// TIA Portal V19 export
FUNCTION_BLOCK "ValveMachine_FB"   // FB125, LAD
TITLE = VALVE MACHINE
// stored: Access Published, MemoryReserve 100, SetENOAutomatically false
   VAR_INPUT
      AreaInterface : "AreaInterface";
      ZSI : "udt_ZoneSafetyInterface";
      DSI : "udt_DeviceSafetyInterface";
      DataIn : "ValveMachine_DataIn";
      Cin : "ValveMachine_Cin";
      Config : "ValveMachine_Config";
   END_VAR
   VAR_OUTPUT
      MachineInterface : "MachineInterface";
      COut : "ValveMachine_COut";
      DataOut : "ValveMachine_DataOut";
   END_VAR
   VAR_IN_OUT
      Alarm : "ValveAlr";
      Warning : "ValveMachine_Wng";
   END_VAR
   VAR
      Sts : Struct
         Standstill : Bool;
         AlarmsPresence : Bool;
         WarningsPresence : Bool;
         Rest_Cnd : Bool;
         Work_Cnd : Bool;
      END_STRUCT;
      Ctrl : Struct
         StopDueDoorOpeningRequest : Bool;
         StopInPhase : Bool;
         StopProgrammed : Bool;
         StopAborting : Bool;
         Work : Bool;
         Rest : Bool;
         Rest_Man : Bool;
         Work_Man : Bool;
         Rest_Aut : Bool;
         Work_Aut : Bool;
      END_STRUCT;
      V : "Valve";
      TON_NoPendingCmd : TON_TIME;
      TON_Rest_MissingExtEnable : TON_TIME;
      TON_Work_MissingExtEnable : TON_TIME;
      TON_PressureRunning_Timeout { S7_SetPoint := 'True'} : TON_TIME;
      Aux : Struct
         Pb_Rest : Bool;
         Pb_Work : Bool;
         Pb_StartStop : Bool;
      END_STRUCT;
   END_VAR
   VAR_TEMP
      PE : Struct
         Pb_Rest : Bool;
         Pb_Work : Bool;
         Pb_StartStop : Bool;
      END_STRUCT;
   END_VAR
   VAR_TEMP   // added for the SCL form of the ladder/FBD networks
      _w1 : Bool;
      _w2 : Bool;
      _w3 : Bool;
   END_VAR
BEGIN

REGION Network 1: Positive edges
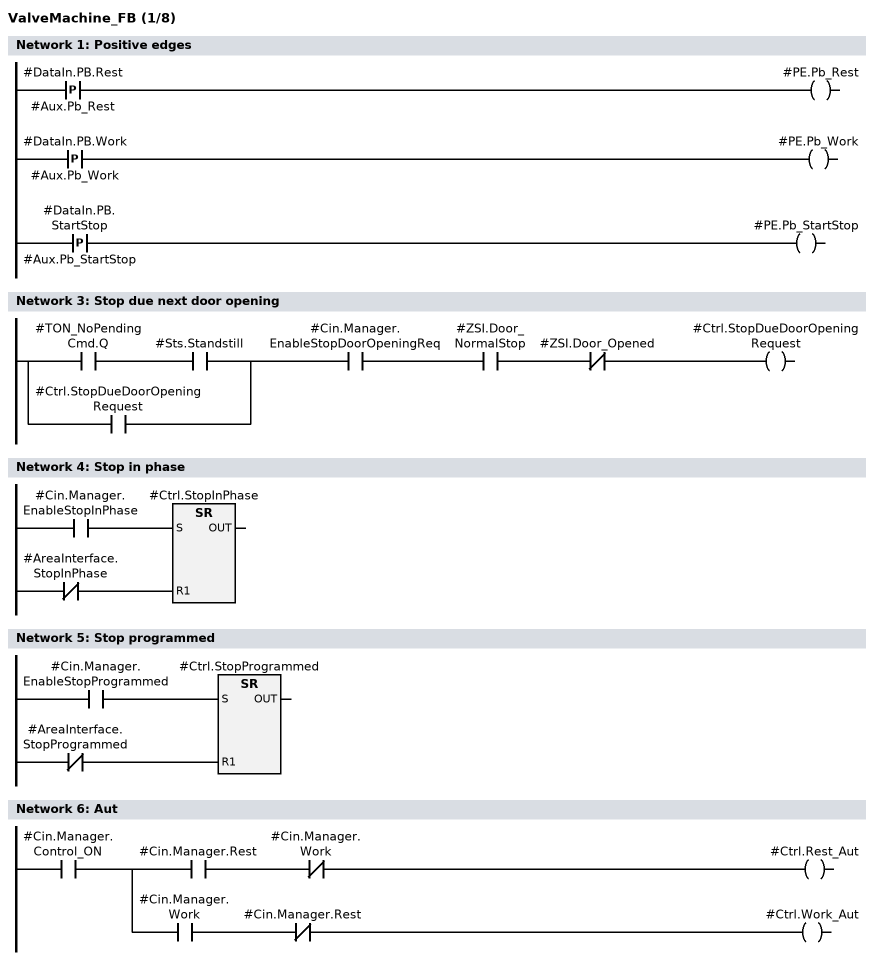
   RUNG wire#powerrail
      P_Contact(operand := #DataIn.PB.Rest, bit := #Aux.Pb_Rest)
      Coil( #PE.Pb_Rest )
   END_RUNG
   RUNG wire#powerrail
      P_Contact(operand := #DataIn.PB.Work, bit := #Aux.Pb_Work)
      Coil( #PE.Pb_Work )
   END_RUNG
   RUNG wire#powerrail
      P_Contact(operand := #DataIn.PB.StartStop, bit := #Aux.Pb_StartStop)
      Coil( #PE.Pb_StartStop )
   END_RUNG
   // the same network as SCL:
   #_w1 := #DataIn.PB.Rest AND NOT #Aux.Pb_Rest;   // rising edge of #DataIn.PB.Rest
   #Aux.Pb_Rest := #DataIn.PB.Rest;
   #PE.Pb_Rest := #_w1;
   #_w2 := #DataIn.PB.Work AND NOT #Aux.Pb_Work;   // rising edge of #DataIn.PB.Work
   #Aux.Pb_Work := #DataIn.PB.Work;
   #PE.Pb_Work := #_w2;
   #_w3 := #DataIn.PB.StartStop AND NOT #Aux.Pb_StartStop;   // rising edge of #DataIn.PB.StartStop
   #Aux.Pb_StartStop := #DataIn.PB.StartStop;
   #PE.Pb_StartStop := #_w3;
END_REGION

REGION Network 2: <<< MACHINE STOP >>>
END_REGION

REGION Network 3: Stop due next door opening
   RUNG wire#powerrail
      Contact( #TON_NoPendingCmd.Q )
      Contact( #Sts.Standstill )
      wire#w1
      Contact( #Cin.Manager.EnableStopDoorOpeningReq )
      Contact( #ZSI.Door_NormalStop )
      I_Contact( #ZSI.Door_Opened )
      Coil( #Ctrl.StopDueDoorOpeningRequest )
   END_RUNG
   RUNG wire#powerrail
      Contact( #Ctrl.StopDueDoorOpeningRequest )
   END_RUNG wire#w1
   // the same network as SCL:
   #Ctrl.StopDueDoorOpeningRequest := ((#TON_NoPendingCmd.Q AND #Sts.Standstill) OR #Ctrl.StopDueDoorOpeningRequest) AND #Cin.Manager.EnableStopDoorOpeningReq AND #ZSI.Door_NormalStop AND NOT #ZSI.Door_Opened;
END_REGION

REGION Network 4: Stop in phase
   RUNG wire#powerrail
      Contact( #Cin.Manager.EnableStopInPhase )
      S_SR(operand := #Ctrl.StopInPhase, r1 := wire#w1)
   END_RUNG
   RUNG wire#powerrail
      I_Contact( #AreaInterface.StopInPhase )
   END_RUNG wire#w1
   // the same network as SCL:
   IF #Cin.Manager.EnableStopInPhase THEN
       #Ctrl.StopInPhase := TRUE;   // SR flip-flop
   END_IF;
   IF NOT #AreaInterface.StopInPhase THEN #Ctrl.StopInPhase := FALSE; END_IF;
END_REGION

REGION Network 5: Stop programmed
   RUNG wire#powerrail
      Contact( #Cin.Manager.EnableStopProgrammed )
      S_SR(operand := #Ctrl.StopProgrammed, r1 := wire#w1)
   END_RUNG
   RUNG wire#powerrail
      I_Contact( #AreaInterface.StopProgrammed )
   END_RUNG wire#w1
   // the same network as SCL:
   IF #Cin.Manager.EnableStopProgrammed THEN
       #Ctrl.StopProgrammed := TRUE;   // SR flip-flop
   END_IF;
   IF NOT #AreaInterface.StopProgrammed THEN #Ctrl.StopProgrammed := FALSE; END_IF;
END_REGION

REGION Network 6: Aut
   RUNG wire#powerrail
      Contact( #Cin.Manager.Control_ON )
      wire#w1
      Contact( #Cin.Manager.Rest )
      I_Contact( #Cin.Manager.Work )
      Coil( #Ctrl.Rest_Aut )
   END_RUNG
   RUNG wire#w1
      Contact( #Cin.Manager.Work )
      I_Contact( #Cin.Manager.Rest )
      Coil( #Ctrl.Work_Aut )
   END_RUNG
   // the same network as SCL:
   #Ctrl.Rest_Aut := #Cin.Manager.Control_ON AND #Cin.Manager.Rest AND NOT #Cin.Manager.Work;
   #Ctrl.Work_Aut := #Cin.Manager.Control_ON AND #Cin.Manager.Work AND NOT #Cin.Manager.Rest;
END_REGION

REGION Network 7: Man
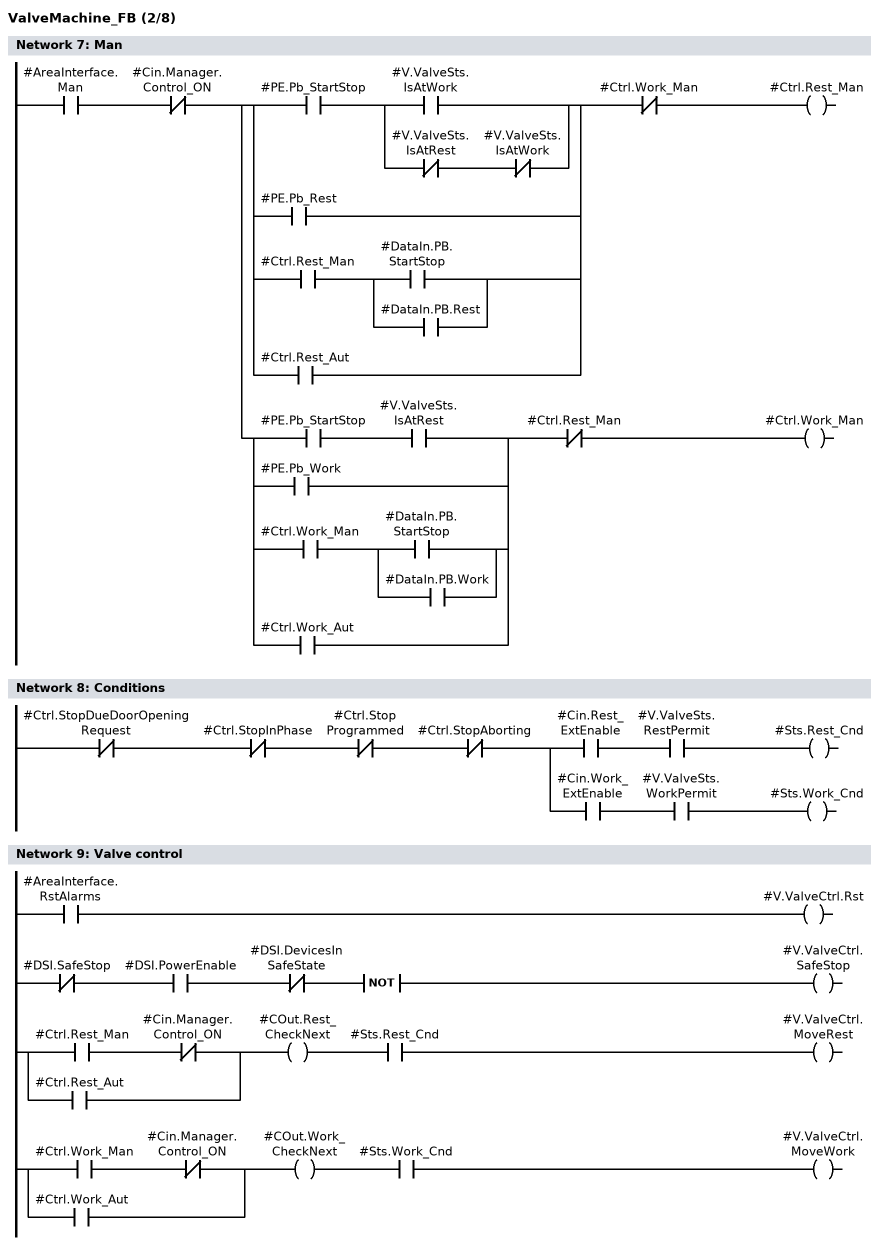
   RUNG wire#powerrail
      Contact( #AreaInterface.Man )
      I_Contact( #Cin.Manager.Control_ON )
      wire#w1
      Contact( #PE.Pb_StartStop )
      wire#w2
      Contact( #V.ValveSts.IsAtWork )
      wire#w3
      I_Contact( #Ctrl.Work_Man )
      Coil( #Ctrl.Rest_Man )
   END_RUNG
   RUNG wire#w2
      I_Contact( #V.ValveSts.IsAtRest )
      I_Contact( #V.ValveSts.IsAtWork )
   END_RUNG wire#w3
   RUNG wire#w1
      Contact( #PE.Pb_Rest )
   END_RUNG wire#w3
   RUNG wire#w1
      Contact( #Ctrl.Rest_Man )
      wire#w4
      Contact( #DataIn.PB.StartStop )
   END_RUNG wire#w3
   RUNG wire#w4
      Contact( #DataIn.PB.Rest )
   END_RUNG wire#w3
   RUNG wire#w1
      Contact( #Ctrl.Rest_Aut )
   END_RUNG wire#w3
   RUNG wire#w1
      Contact( #PE.Pb_StartStop )
      Contact( #V.ValveSts.IsAtRest )
      wire#w5
      I_Contact( #Ctrl.Rest_Man )
      Coil( #Ctrl.Work_Man )
   END_RUNG
   RUNG wire#w1
      Contact( #PE.Pb_Work )
   END_RUNG wire#w5
   RUNG wire#w1
      Contact( #Ctrl.Work_Man )
      wire#w6
      Contact( #DataIn.PB.StartStop )
   END_RUNG wire#w5
   RUNG wire#w6
      Contact( #DataIn.PB.Work )
   END_RUNG wire#w5
   RUNG wire#w1
      Contact( #Ctrl.Work_Aut )
   END_RUNG wire#w5
   // the same network as SCL:
   #_w1 := #AreaInterface.Man AND NOT #Cin.Manager.Control_ON;
   #Ctrl.Rest_Man := #_w1 AND ((#PE.Pb_StartStop AND (#V.ValveSts.IsAtWork OR (NOT #V.ValveSts.IsAtRest AND NOT #V.ValveSts.IsAtWork))) OR #PE.Pb_Rest OR (#Ctrl.Rest_Man AND (#DataIn.PB.StartStop OR #DataIn.PB.Rest)) OR #Ctrl.Rest_Aut) AND NOT #Ctrl.Work_Man;
   #Ctrl.Work_Man := #_w1 AND ((#PE.Pb_StartStop AND #V.ValveSts.IsAtRest) OR #PE.Pb_Work OR (#Ctrl.Work_Man AND (#DataIn.PB.StartStop OR #DataIn.PB.Work)) OR #Ctrl.Work_Aut) AND NOT #Ctrl.Rest_Man;
END_REGION

REGION Network 8: Conditions
   RUNG wire#powerrail
      I_Contact( #Ctrl.StopDueDoorOpeningRequest )
      I_Contact( #Ctrl.StopInPhase )
      I_Contact( #Ctrl.StopProgrammed )
      I_Contact( #Ctrl.StopAborting )
      wire#w1
      Contact( #Cin.Rest_ExtEnable )
      Contact( #V.ValveSts.RestPermit )
      Coil( #Sts.Rest_Cnd )
   END_RUNG
   RUNG wire#w1
      Contact( #Cin.Work_ExtEnable )
      Contact( #V.ValveSts.WorkPermit )
      Coil( #Sts.Work_Cnd )
   END_RUNG
   // the same network as SCL:
   #_w1 := NOT #Ctrl.StopDueDoorOpeningRequest AND NOT #Ctrl.StopInPhase AND NOT #Ctrl.StopProgrammed AND NOT #Ctrl.StopAborting;
   #Sts.Rest_Cnd := #_w1 AND #Cin.Rest_ExtEnable AND #V.ValveSts.RestPermit;
   #Sts.Work_Cnd := #_w1 AND #Cin.Work_ExtEnable AND #V.ValveSts.WorkPermit;
END_REGION

REGION Network 9: Valve control
   RUNG wire#powerrail
      Contact( #AreaInterface.RstAlarms )
      Coil( #V.ValveCtrl.Rst )
   END_RUNG
   RUNG wire#powerrail
      I_Contact( #DSI.SafeStop )
      Contact( #DSI.PowerEnable )
      I_Contact( #DSI.DevicesInSafeState )
      Not()
      Coil( #V.ValveCtrl.SafeStop )
   END_RUNG
   RUNG wire#powerrail
      Contact( #Ctrl.Rest_Man )
      I_Contact( #Cin.Manager.Control_ON )
      wire#w1
      Coil( #COut.Rest_CheckNext )
      Contact( #Sts.Rest_Cnd )
      Coil( #V.ValveCtrl.MoveRest )
   END_RUNG
   RUNG wire#powerrail
      Contact( #Ctrl.Rest_Aut )
   END_RUNG wire#w1
   RUNG wire#powerrail
      Contact( #Ctrl.Work_Man )
      I_Contact( #Cin.Manager.Control_ON )
      wire#w2
      Coil( #COut.Work_CheckNext )
      Contact( #Sts.Work_Cnd )
      Coil( #V.ValveCtrl.MoveWork )
   END_RUNG
   RUNG wire#powerrail
      Contact( #Ctrl.Work_Aut )
   END_RUNG wire#w2
   // the same network as SCL:
   #V.ValveCtrl.Rst := #AreaInterface.RstAlarms;
   #V.ValveCtrl.SafeStop := NOT (NOT #DSI.SafeStop AND #DSI.PowerEnable AND NOT #DSI.DevicesInSafeState);
   #COut.Rest_CheckNext := (#Ctrl.Rest_Man AND NOT #Cin.Manager.Control_ON) OR #Ctrl.Rest_Aut;
   #V.ValveCtrl.MoveRest := #COut.Rest_CheckNext AND #Sts.Rest_Cnd;
   #COut.Work_CheckNext := (#Ctrl.Work_Man AND NOT #Cin.Manager.Control_ON) OR #Ctrl.Work_Aut;
   #V.ValveCtrl.MoveWork := #COut.Work_CheckNext AND #Sts.Work_Cnd;
END_REGION

REGION Network 10: Warning missing external enables
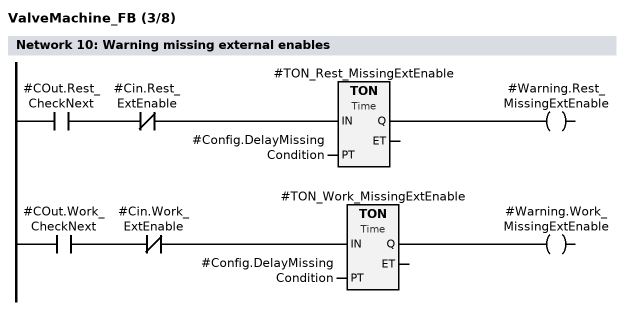
   RUNG wire#powerrail
      Contact( #COut.Rest_CheckNext )
      I_Contact( #Cin.Rest_ExtEnable )
      { S7_Templates := "time_type := Time" } #TON_Rest_MissingExtEnable.TON(pt := #Config.DelayMissingCondition, et =>)
      Coil( #Warning.Rest_MissingExtEnable )
   END_RUNG
   RUNG wire#powerrail
      Contact( #COut.Work_CheckNext )
      I_Contact( #Cin.Work_ExtEnable )
      { S7_Templates := "time_type := Time" } #TON_Work_MissingExtEnable.TON(pt := #Config.DelayMissingCondition, et =>)
      Coil( #Warning.Work_MissingExtEnable )
   END_RUNG
   // the same network as SCL:
   #TON_Rest_MissingExtEnable(IN := #COut.Rest_CheckNext AND NOT #Cin.Rest_ExtEnable,   // TON
                           PT := #Config.DelayMissingCondition);
   #Warning.Rest_MissingExtEnable := #TON_Rest_MissingExtEnable.Q;
   #TON_Work_MissingExtEnable(IN := #COut.Work_CheckNext AND NOT #Cin.Work_ExtEnable,   // TON
                           PT := #Config.DelayMissingCondition);
   #Warning.Work_MissingExtEnable := #TON_Work_MissingExtEnable.Q;
END_REGION

REGION Network 11: Valve manager
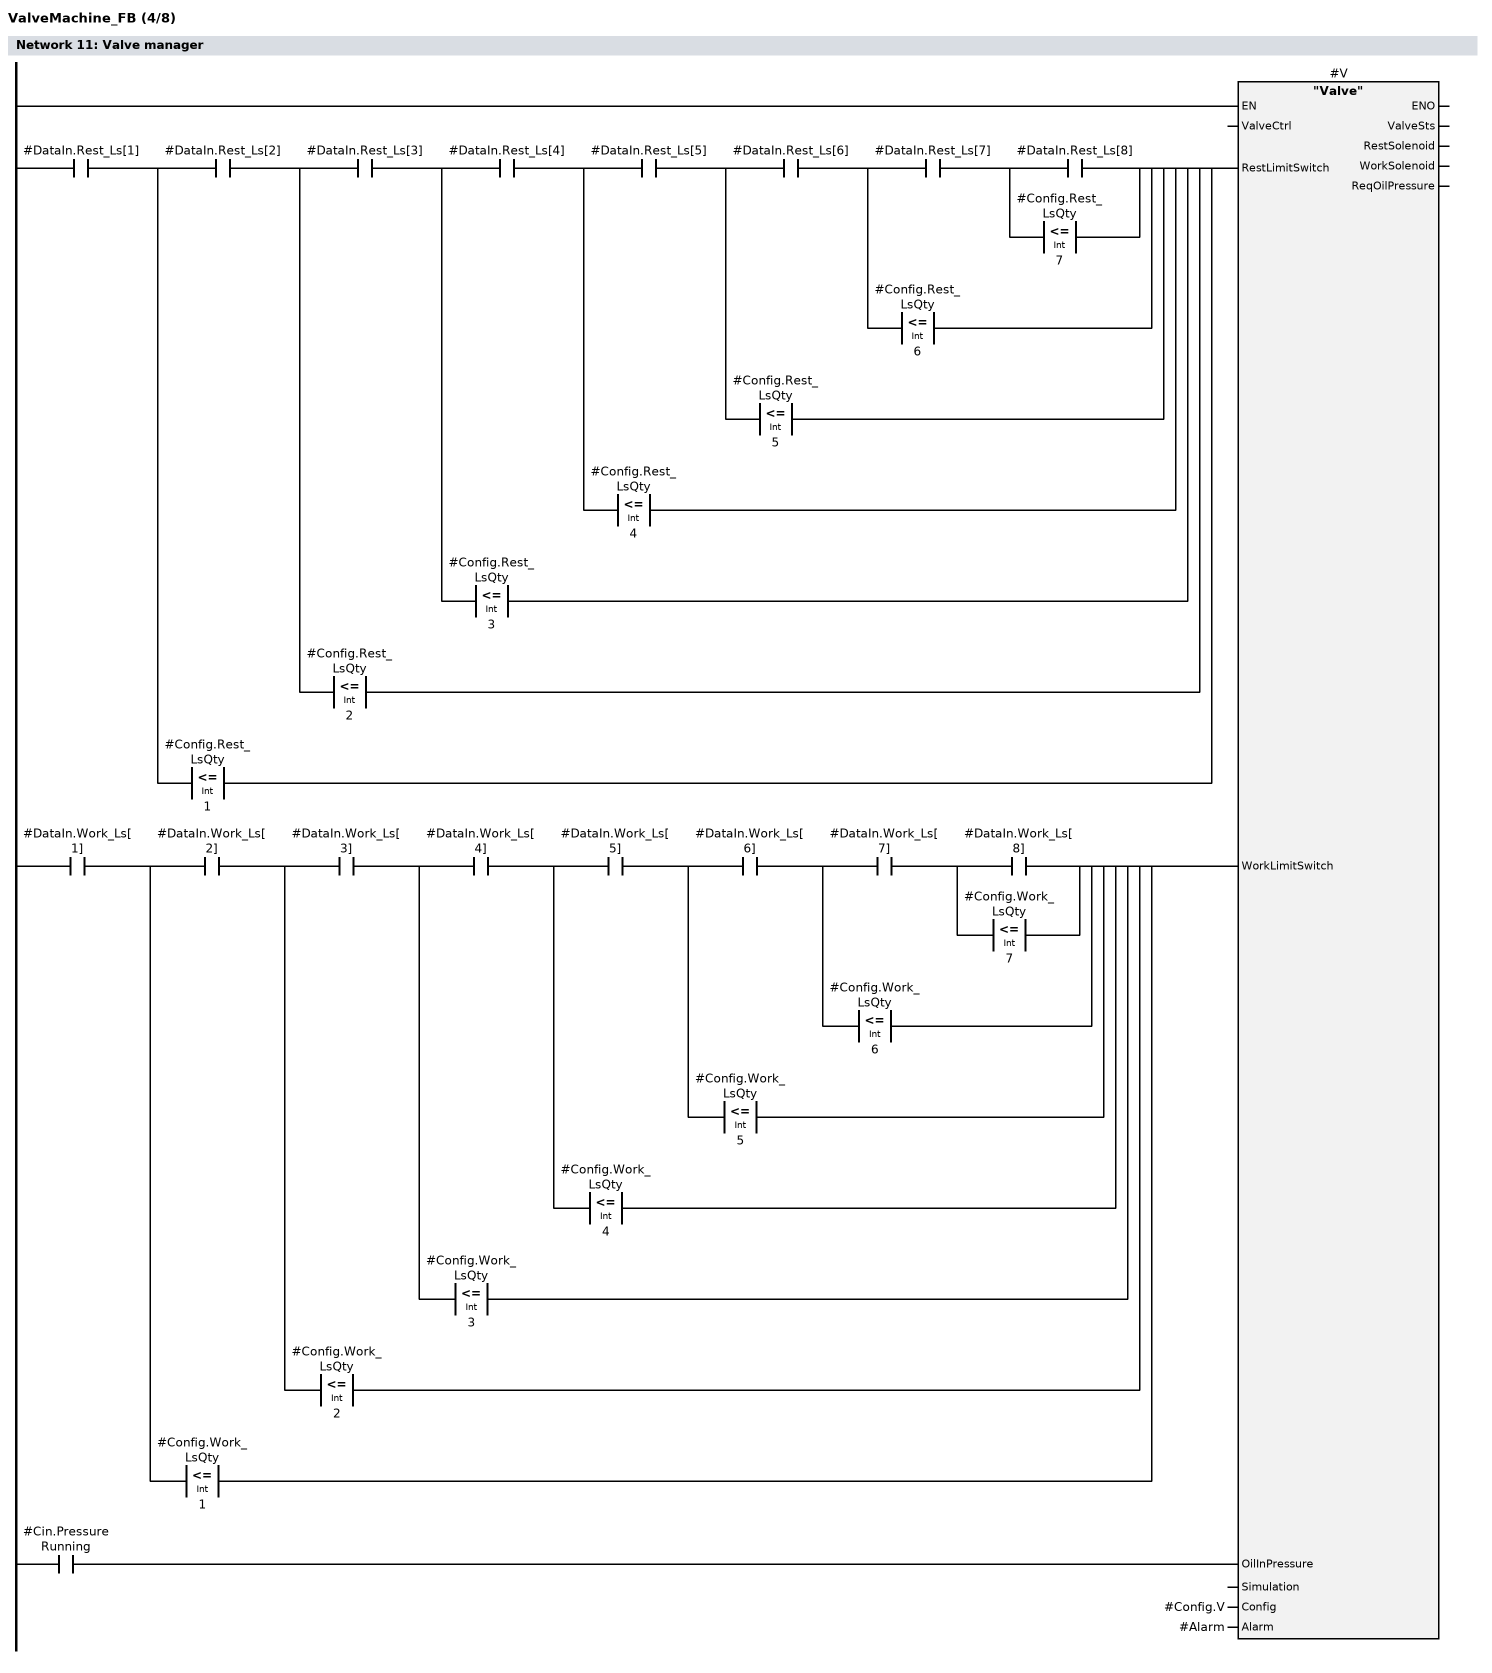
   RUNG wire#powerrail
      #V(RestLimitSwitch := wire#w8, WorkLimitSwitch := wire#w16, OilInPressure := wire#w17, ValveCtrl :=, Simulation :=, Config := #Config.V, Alarm := #Alarm, ValveSts =>, RestSolenoid =>, WorkSolenoid =>, ReqOilPressure =>)
   END_RUNG
   RUNG wire#powerrail
      Contact( #DataIn.Rest_Ls[1] )
      wire#w1
      Contact( #DataIn.Rest_Ls[2] )
      wire#w2
      Contact( #DataIn.Rest_Ls[3] )
      wire#w3
      Contact( #DataIn.Rest_Ls[4] )
      wire#w4
      Contact( #DataIn.Rest_Ls[5] )
      wire#w5
      Contact( #DataIn.Rest_Ls[6] )
      wire#w6
      Contact( #DataIn.Rest_Ls[7] )
      wire#w7
      Contact( #DataIn.Rest_Ls[8] )
   END_RUNG wire#w8
   RUNG wire#w7
      { S7_Templates := "SrcType := Int" } LE_Contact(in1 := #Config.Rest_LsQty, in2 := 7)
   END_RUNG wire#w8
   RUNG wire#w6
      { S7_Templates := "SrcType := Int" } LE_Contact(in1 := #Config.Rest_LsQty, in2 := 6)
   END_RUNG wire#w8
   RUNG wire#w5
      { S7_Templates := "SrcType := Int" } LE_Contact(in1 := #Config.Rest_LsQty, in2 := 5)
   END_RUNG wire#w8
   RUNG wire#w4
      { S7_Templates := "SrcType := Int" } LE_Contact(in1 := #Config.Rest_LsQty, in2 := 4)
   END_RUNG wire#w8
   RUNG wire#w3
      { S7_Templates := "SrcType := Int" } LE_Contact(in1 := #Config.Rest_LsQty, in2 := 3)
   END_RUNG wire#w8
   RUNG wire#w2
      { S7_Templates := "SrcType := Int" } LE_Contact(in1 := #Config.Rest_LsQty, in2 := 2)
   END_RUNG wire#w8
   RUNG wire#w1
      { S7_Templates := "SrcType := Int" } LE_Contact(in1 := #Config.Rest_LsQty, in2 := 1)
   END_RUNG wire#w8
   RUNG wire#powerrail
      Contact( #DataIn.Work_Ls[1] )
      wire#w9
      Contact( #DataIn.Work_Ls[2] )
      wire#w10
      Contact( #DataIn.Work_Ls[3] )
      wire#w11
      Contact( #DataIn.Work_Ls[4] )
      wire#w12
      Contact( #DataIn.Work_Ls[5] )
      wire#w13
      Contact( #DataIn.Work_Ls[6] )
      wire#w14
      Contact( #DataIn.Work_Ls[7] )
      wire#w15
      Contact( #DataIn.Work_Ls[8] )
   END_RUNG wire#w16
   RUNG wire#w15
      { S7_Templates := "SrcType := Int" } LE_Contact(in1 := #Config.Work_LsQty, in2 := 7)
   END_RUNG wire#w16
   RUNG wire#w14
      { S7_Templates := "SrcType := Int" } LE_Contact(in1 := #Config.Work_LsQty, in2 := 6)
   END_RUNG wire#w16
   RUNG wire#w13
      { S7_Templates := "SrcType := Int" } LE_Contact(in1 := #Config.Work_LsQty, in2 := 5)
   END_RUNG wire#w16
   RUNG wire#w12
      { S7_Templates := "SrcType := Int" } LE_Contact(in1 := #Config.Work_LsQty, in2 := 4)
   END_RUNG wire#w16
   RUNG wire#w11
      { S7_Templates := "SrcType := Int" } LE_Contact(in1 := #Config.Work_LsQty, in2 := 3)
   END_RUNG wire#w16
   RUNG wire#w10
      { S7_Templates := "SrcType := Int" } LE_Contact(in1 := #Config.Work_LsQty, in2 := 2)
   END_RUNG wire#w16
   RUNG wire#w9
      { S7_Templates := "SrcType := Int" } LE_Contact(in1 := #Config.Work_LsQty, in2 := 1)
   END_RUNG wire#w16
   RUNG wire#powerrail
      Contact( #Cin.PressureRunning )
   END_RUNG wire#w17
   // the same network as SCL:
   #V(RestLimitSwitch := #DataIn.Rest_Ls[1] AND ((#DataIn.Rest_Ls[2] AND ((#DataIn.Rest_Ls[3] AND ((#DataIn.Rest_Ls[4] AND ((#DataIn.Rest_Ls[5] AND ((#DataIn.Rest_Ls[6] AND ((#DataIn.Rest_Ls[7] AND (#DataIn.Rest_Ls[8] OR (#Config.Rest_LsQty <= 7))) OR (#Config.Rest_LsQty <= 6))) OR (#Config.Rest_LsQty <= 5))) OR (#Config.Rest_LsQty <= 4))) OR (#Config.Rest_LsQty <= 3))) OR (#Config.Rest_LsQty <= 2))) OR (#Config.Rest_LsQty <= 1)),   // "Valve"
      WorkLimitSwitch := #DataIn.Work_Ls[1] AND ((#DataIn.Work_Ls[2] AND ((#DataIn.Work_Ls[3] AND ((#DataIn.Work_Ls[4] AND ((#DataIn.Work_Ls[5] AND ((#DataIn.Work_Ls[6] AND ((#DataIn.Work_Ls[7] AND (#DataIn.Work_Ls[8] OR (#Config.Work_LsQty <= 7))) OR (#Config.Work_LsQty <= 6))) OR (#Config.Work_LsQty <= 5))) OR (#Config.Work_LsQty <= 4))) OR (#Config.Work_LsQty <= 3))) OR (#Config.Work_LsQty <= 2))) OR (#Config.Work_LsQty <= 1)),
      OilInPressure := #Cin.PressureRunning,
      Config := #Config.V,
      Alarm := #Alarm);
END_REGION

REGION Network 12: Warning missing REST Ls
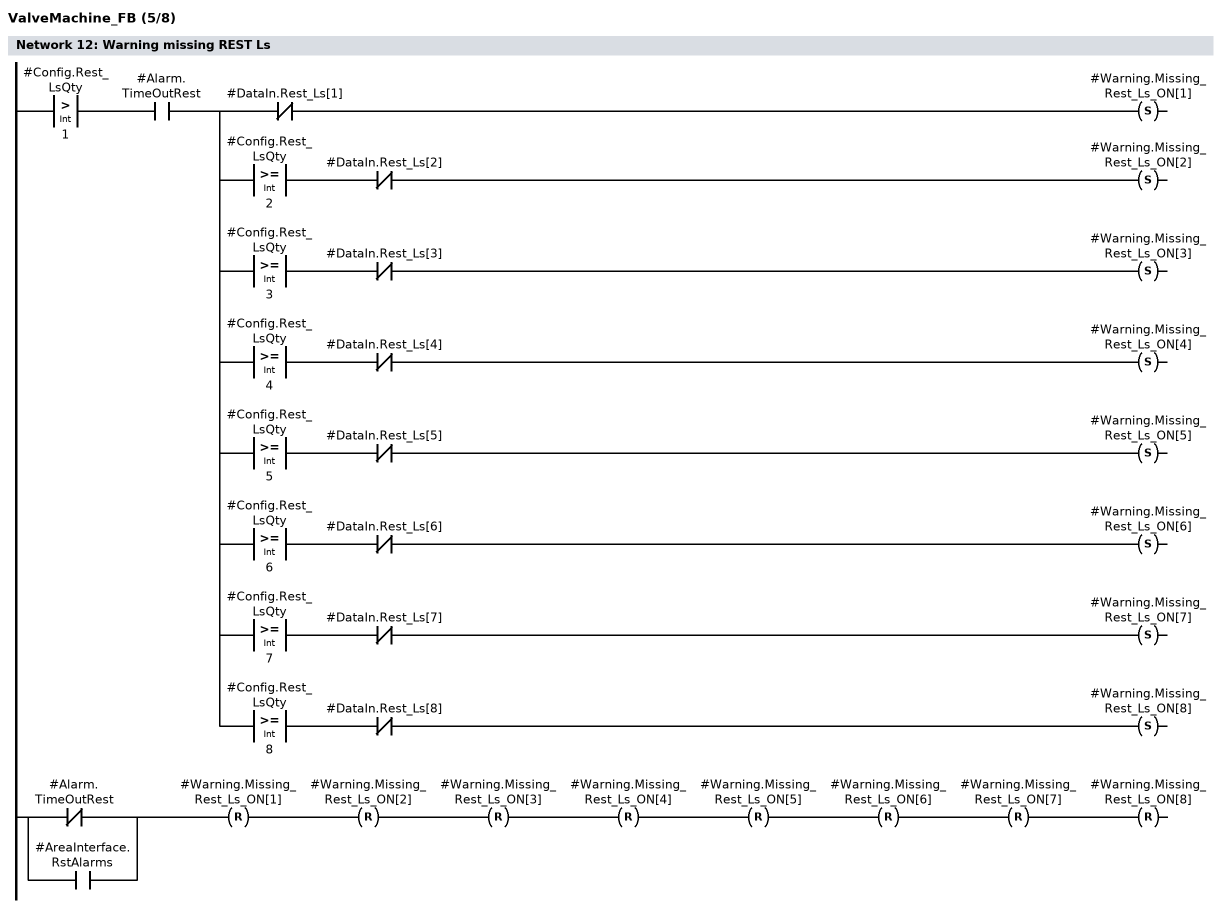
   RUNG wire#powerrail
      { S7_Templates := "SrcType := Int" } GT_Contact(in1 := #Config.Rest_LsQty, in2 := 1)
      Contact( #Alarm.TimeOutRest )
      wire#w1
      I_Contact( #DataIn.Rest_Ls[1] )
      S_Coil( #Warning.Missing_Rest_Ls_ON[1] )
   END_RUNG
   RUNG wire#w1
      { S7_Templates := "SrcType := Int" } GE_Contact(in1 := #Config.Rest_LsQty, in2 := 2)
      I_Contact( #DataIn.Rest_Ls[2] )
      S_Coil( #Warning.Missing_Rest_Ls_ON[2] )
   END_RUNG
   RUNG wire#w1
      { S7_Templates := "SrcType := Int" } GE_Contact(in1 := #Config.Rest_LsQty, in2 := 3)
      I_Contact( #DataIn.Rest_Ls[3] )
      S_Coil( #Warning.Missing_Rest_Ls_ON[3] )
   END_RUNG
   RUNG wire#w1
      { S7_Templates := "SrcType := Int" } GE_Contact(in1 := #Config.Rest_LsQty, in2 := 4)
      I_Contact( #DataIn.Rest_Ls[4] )
      S_Coil( #Warning.Missing_Rest_Ls_ON[4] )
   END_RUNG
   RUNG wire#w1
      { S7_Templates := "SrcType := Int" } GE_Contact(in1 := #Config.Rest_LsQty, in2 := 5)
      I_Contact( #DataIn.Rest_Ls[5] )
      S_Coil( #Warning.Missing_Rest_Ls_ON[5] )
   END_RUNG
   RUNG wire#w1
      { S7_Templates := "SrcType := Int" } GE_Contact(in1 := #Config.Rest_LsQty, in2 := 6)
      I_Contact( #DataIn.Rest_Ls[6] )
      S_Coil( #Warning.Missing_Rest_Ls_ON[6] )
   END_RUNG
   RUNG wire#w1
      { S7_Templates := "SrcType := Int" } GE_Contact(in1 := #Config.Rest_LsQty, in2 := 7)
      I_Contact( #DataIn.Rest_Ls[7] )
      S_Coil( #Warning.Missing_Rest_Ls_ON[7] )
   END_RUNG
   RUNG wire#w1
      { S7_Templates := "SrcType := Int" } GE_Contact(in1 := #Config.Rest_LsQty, in2 := 8)
      I_Contact( #DataIn.Rest_Ls[8] )
      S_Coil( #Warning.Missing_Rest_Ls_ON[8] )
   END_RUNG
   RUNG wire#powerrail
      I_Contact( #Alarm.TimeOutRest )
      wire#w2
      R_Coil( #Warning.Missing_Rest_Ls_ON[1] )
      R_Coil( #Warning.Missing_Rest_Ls_ON[2] )
      R_Coil( #Warning.Missing_Rest_Ls_ON[3] )
      R_Coil( #Warning.Missing_Rest_Ls_ON[4] )
      R_Coil( #Warning.Missing_Rest_Ls_ON[5] )
      R_Coil( #Warning.Missing_Rest_Ls_ON[6] )
      R_Coil( #Warning.Missing_Rest_Ls_ON[7] )
      R_Coil( #Warning.Missing_Rest_Ls_ON[8] )
   END_RUNG
   RUNG wire#powerrail
      Contact( #AreaInterface.RstAlarms )
   END_RUNG wire#w2
   // the same network as SCL:
   #_w1 := (#Config.Rest_LsQty > 1) AND #Alarm.TimeOutRest;
   IF #_w1 AND NOT #DataIn.Rest_Ls[1] THEN #Warning.Missing_Rest_Ls_ON[1] := TRUE; END_IF;
   IF #_w1 AND (#Config.Rest_LsQty >= 2) AND NOT #DataIn.Rest_Ls[2] THEN
       #Warning.Missing_Rest_Ls_ON[2] := TRUE;
   END_IF;
   IF #_w1 AND (#Config.Rest_LsQty >= 3) AND NOT #DataIn.Rest_Ls[3] THEN
       #Warning.Missing_Rest_Ls_ON[3] := TRUE;
   END_IF;
   IF #_w1 AND (#Config.Rest_LsQty >= 4) AND NOT #DataIn.Rest_Ls[4] THEN
       #Warning.Missing_Rest_Ls_ON[4] := TRUE;
   END_IF;
   IF #_w1 AND (#Config.Rest_LsQty >= 5) AND NOT #DataIn.Rest_Ls[5] THEN
       #Warning.Missing_Rest_Ls_ON[5] := TRUE;
   END_IF;
   IF #_w1 AND (#Config.Rest_LsQty >= 6) AND NOT #DataIn.Rest_Ls[6] THEN
       #Warning.Missing_Rest_Ls_ON[6] := TRUE;
   END_IF;
   IF #_w1 AND (#Config.Rest_LsQty >= 7) AND NOT #DataIn.Rest_Ls[7] THEN
       #Warning.Missing_Rest_Ls_ON[7] := TRUE;
   END_IF;
   IF #_w1 AND (#Config.Rest_LsQty >= 8) AND NOT #DataIn.Rest_Ls[8] THEN
       #Warning.Missing_Rest_Ls_ON[8] := TRUE;
   END_IF;
   IF NOT #Alarm.TimeOutRest OR #AreaInterface.RstAlarms THEN
       #Warning.Missing_Rest_Ls_ON[1] := FALSE;
       #Warning.Missing_Rest_Ls_ON[2] := FALSE;
       #Warning.Missing_Rest_Ls_ON[3] := FALSE;
       #Warning.Missing_Rest_Ls_ON[4] := FALSE;
       #Warning.Missing_Rest_Ls_ON[5] := FALSE;
       #Warning.Missing_Rest_Ls_ON[6] := FALSE;
       #Warning.Missing_Rest_Ls_ON[7] := FALSE;
       #Warning.Missing_Rest_Ls_ON[8] := FALSE;
   END_IF;
END_REGION

REGION Network 13: Warning missing WORK Ls
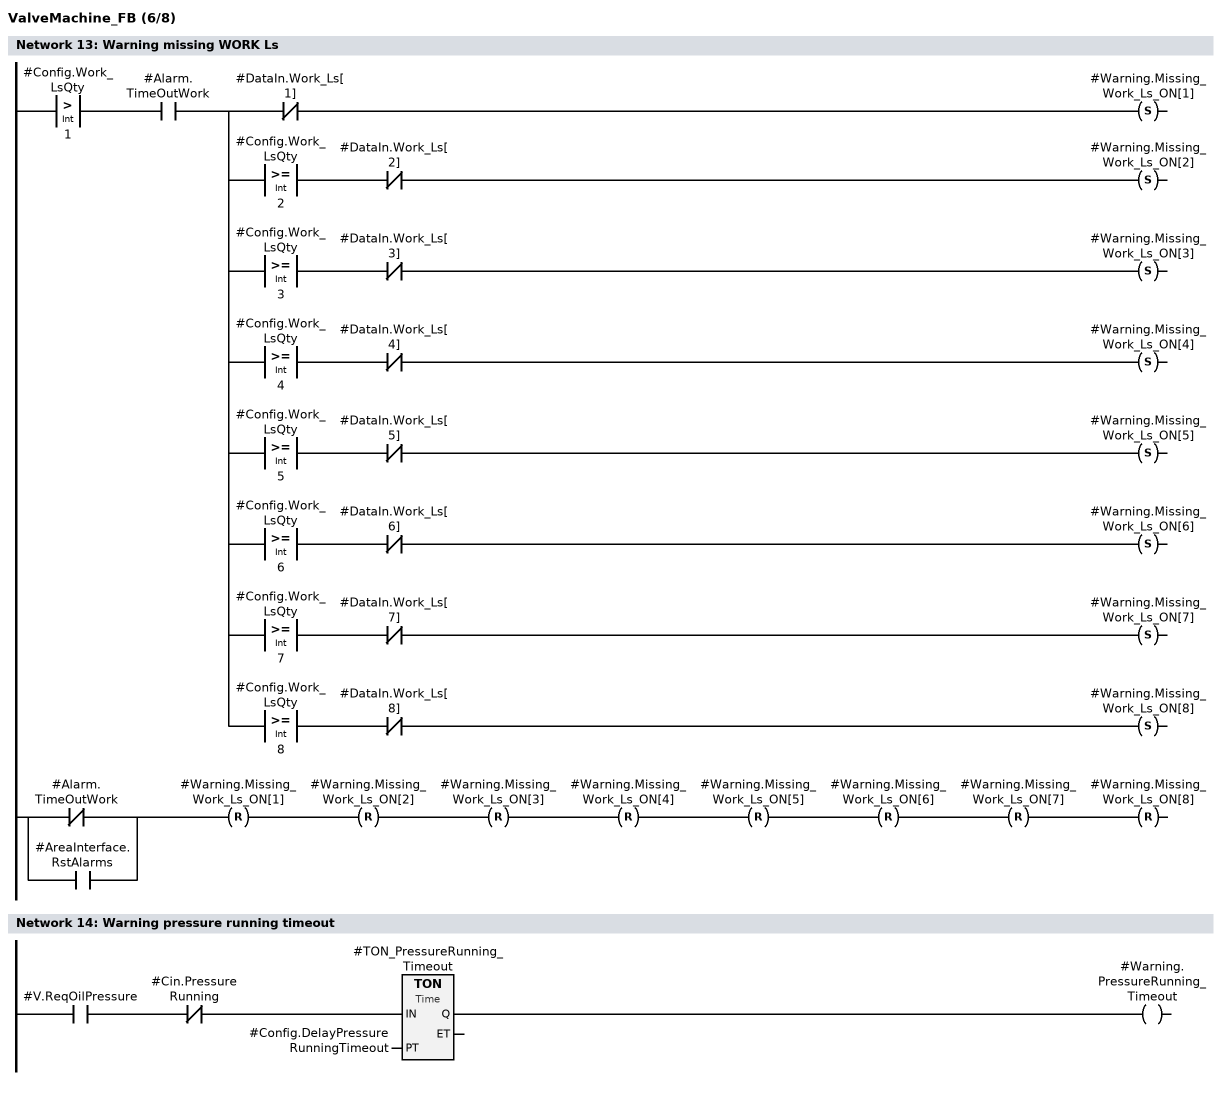
   RUNG wire#powerrail
      { S7_Templates := "SrcType := Int" } GT_Contact(in1 := #Config.Work_LsQty, in2 := 1)
      Contact( #Alarm.TimeOutWork )
      wire#w1
      I_Contact( #DataIn.Work_Ls[1] )
      S_Coil( #Warning.Missing_Work_Ls_ON[1] )
   END_RUNG
   RUNG wire#w1
      { S7_Templates := "SrcType := Int" } GE_Contact(in1 := #Config.Work_LsQty, in2 := 2)
      I_Contact( #DataIn.Work_Ls[2] )
      S_Coil( #Warning.Missing_Work_Ls_ON[2] )
   END_RUNG
   RUNG wire#w1
      { S7_Templates := "SrcType := Int" } GE_Contact(in1 := #Config.Work_LsQty, in2 := 3)
      I_Contact( #DataIn.Work_Ls[3] )
      S_Coil( #Warning.Missing_Work_Ls_ON[3] )
   END_RUNG
   RUNG wire#w1
      { S7_Templates := "SrcType := Int" } GE_Contact(in1 := #Config.Work_LsQty, in2 := 4)
      I_Contact( #DataIn.Work_Ls[4] )
      S_Coil( #Warning.Missing_Work_Ls_ON[4] )
   END_RUNG
   RUNG wire#w1
      { S7_Templates := "SrcType := Int" } GE_Contact(in1 := #Config.Work_LsQty, in2 := 5)
      I_Contact( #DataIn.Work_Ls[5] )
      S_Coil( #Warning.Missing_Work_Ls_ON[5] )
   END_RUNG
   RUNG wire#w1
      { S7_Templates := "SrcType := Int" } GE_Contact(in1 := #Config.Work_LsQty, in2 := 6)
      I_Contact( #DataIn.Work_Ls[6] )
      S_Coil( #Warning.Missing_Work_Ls_ON[6] )
   END_RUNG
   RUNG wire#w1
      { S7_Templates := "SrcType := Int" } GE_Contact(in1 := #Config.Work_LsQty, in2 := 7)
      I_Contact( #DataIn.Work_Ls[7] )
      S_Coil( #Warning.Missing_Work_Ls_ON[7] )
   END_RUNG
   RUNG wire#w1
      { S7_Templates := "SrcType := Int" } GE_Contact(in1 := #Config.Work_LsQty, in2 := 8)
      I_Contact( #DataIn.Work_Ls[8] )
      S_Coil( #Warning.Missing_Work_Ls_ON[8] )
   END_RUNG
   RUNG wire#powerrail
      I_Contact( #Alarm.TimeOutWork )
      wire#w2
      R_Coil( #Warning.Missing_Work_Ls_ON[1] )
      R_Coil( #Warning.Missing_Work_Ls_ON[2] )
      R_Coil( #Warning.Missing_Work_Ls_ON[3] )
      R_Coil( #Warning.Missing_Work_Ls_ON[4] )
      R_Coil( #Warning.Missing_Work_Ls_ON[5] )
      R_Coil( #Warning.Missing_Work_Ls_ON[6] )
      R_Coil( #Warning.Missing_Work_Ls_ON[7] )
      R_Coil( #Warning.Missing_Work_Ls_ON[8] )
   END_RUNG
   RUNG wire#powerrail
      Contact( #AreaInterface.RstAlarms )
   END_RUNG wire#w2
   // the same network as SCL:
   #_w1 := (#Config.Work_LsQty > 1) AND #Alarm.TimeOutWork;
   IF #_w1 AND NOT #DataIn.Work_Ls[1] THEN #Warning.Missing_Work_Ls_ON[1] := TRUE; END_IF;
   IF #_w1 AND (#Config.Work_LsQty >= 2) AND NOT #DataIn.Work_Ls[2] THEN
       #Warning.Missing_Work_Ls_ON[2] := TRUE;
   END_IF;
   IF #_w1 AND (#Config.Work_LsQty >= 3) AND NOT #DataIn.Work_Ls[3] THEN
       #Warning.Missing_Work_Ls_ON[3] := TRUE;
   END_IF;
   IF #_w1 AND (#Config.Work_LsQty >= 4) AND NOT #DataIn.Work_Ls[4] THEN
       #Warning.Missing_Work_Ls_ON[4] := TRUE;
   END_IF;
   IF #_w1 AND (#Config.Work_LsQty >= 5) AND NOT #DataIn.Work_Ls[5] THEN
       #Warning.Missing_Work_Ls_ON[5] := TRUE;
   END_IF;
   IF #_w1 AND (#Config.Work_LsQty >= 6) AND NOT #DataIn.Work_Ls[6] THEN
       #Warning.Missing_Work_Ls_ON[6] := TRUE;
   END_IF;
   IF #_w1 AND (#Config.Work_LsQty >= 7) AND NOT #DataIn.Work_Ls[7] THEN
       #Warning.Missing_Work_Ls_ON[7] := TRUE;
   END_IF;
   IF #_w1 AND (#Config.Work_LsQty >= 8) AND NOT #DataIn.Work_Ls[8] THEN
       #Warning.Missing_Work_Ls_ON[8] := TRUE;
   END_IF;
   IF NOT #Alarm.TimeOutWork OR #AreaInterface.RstAlarms THEN
       #Warning.Missing_Work_Ls_ON[1] := FALSE;
       #Warning.Missing_Work_Ls_ON[2] := FALSE;
       #Warning.Missing_Work_Ls_ON[3] := FALSE;
       #Warning.Missing_Work_Ls_ON[4] := FALSE;
       #Warning.Missing_Work_Ls_ON[5] := FALSE;
       #Warning.Missing_Work_Ls_ON[6] := FALSE;
       #Warning.Missing_Work_Ls_ON[7] := FALSE;
       #Warning.Missing_Work_Ls_ON[8] := FALSE;
   END_IF;
END_REGION

REGION Network 14: Warning pressure running timeout
   RUNG wire#powerrail
      Contact( #V.ReqOilPressure )
      I_Contact( #Cin.PressureRunning )
      { S7_Templates := "time_type := Time" } #TON_PressureRunning_Timeout.TON(pt := #Config.DelayPressureRunningTimeout, et =>)
      Coil( #Warning.PressureRunning_Timeout )
   END_RUNG
   // the same network as SCL:
   #TON_PressureRunning_Timeout(IN := #V.ReqOilPressure AND NOT #Cin.PressureRunning,   // TON
                           PT := #Config.DelayPressureRunningTimeout);
   #Warning.PressureRunning_Timeout := #TON_PressureRunning_Timeout.Q;
END_REGION

REGION Network 15: Coordination out
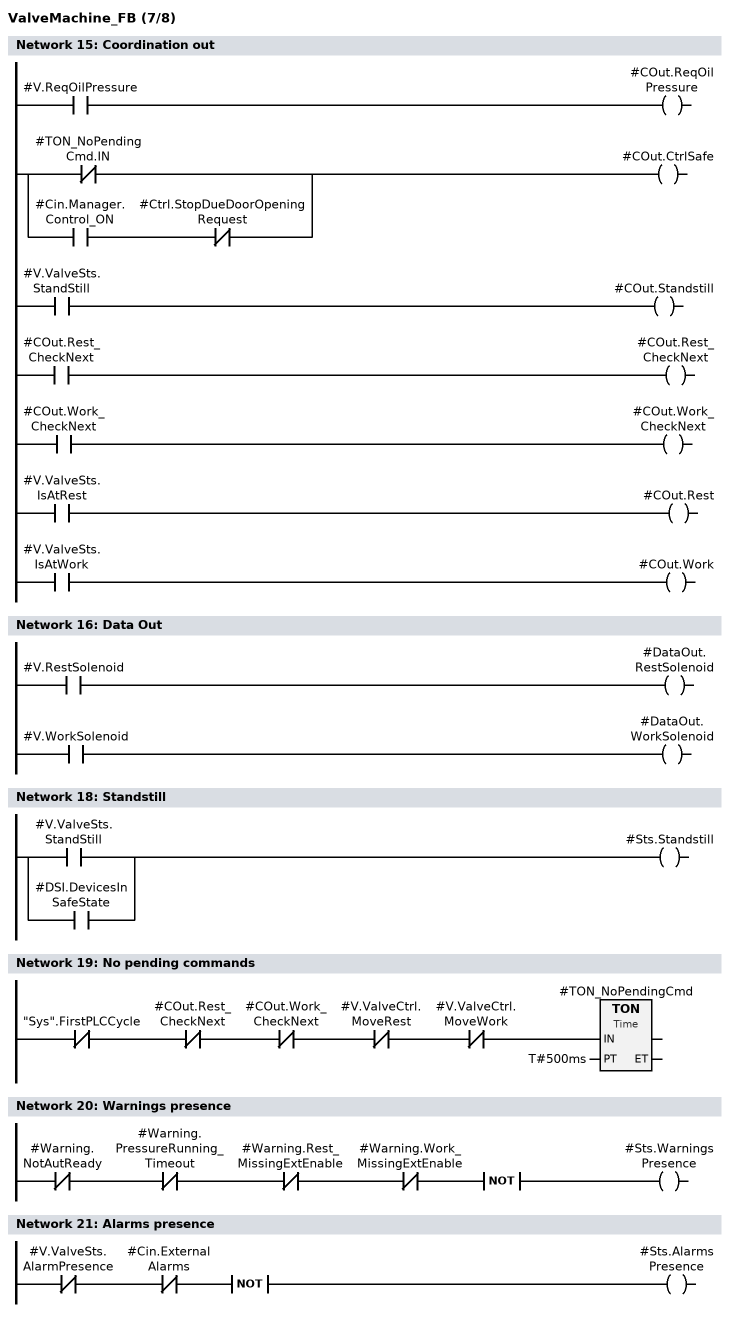
   RUNG wire#powerrail
      Contact( #V.ReqOilPressure )
      Coil( #COut.ReqOilPressure )
   END_RUNG
   RUNG wire#powerrail
      I_Contact( #TON_NoPendingCmd.IN )
      wire#w1
      Coil( #COut.CtrlSafe )
   END_RUNG
   RUNG wire#powerrail
      Contact( #Cin.Manager.Control_ON )
      I_Contact( #Ctrl.StopDueDoorOpeningRequest )
   END_RUNG wire#w1
   RUNG wire#powerrail
      Contact( #V.ValveSts.StandStill )
      Coil( #COut.Standstill )
   END_RUNG
   RUNG wire#powerrail
      Contact( #COut.Rest_CheckNext )
      Coil( #COut.Rest_CheckNext )
   END_RUNG
   RUNG wire#powerrail
      Contact( #COut.Work_CheckNext )
      Coil( #COut.Work_CheckNext )
   END_RUNG
   RUNG wire#powerrail
      Contact( #V.ValveSts.IsAtRest )
      Coil( #COut.Rest )
   END_RUNG
   RUNG wire#powerrail
      Contact( #V.ValveSts.IsAtWork )
      Coil( #COut.Work )
   END_RUNG
   // the same network as SCL:
   #COut.ReqOilPressure := #V.ReqOilPressure;
   #COut.CtrlSafe := NOT #TON_NoPendingCmd.IN OR (#Cin.Manager.Control_ON AND NOT #Ctrl.StopDueDoorOpeningRequest);
   #COut.Standstill := #V.ValveSts.StandStill;
   #COut.Rest_CheckNext := #COut.Rest_CheckNext;
   #COut.Work_CheckNext := #COut.Work_CheckNext;
   #COut.Rest := #V.ValveSts.IsAtRest;
   #COut.Work := #V.ValveSts.IsAtWork;
END_REGION

REGION Network 16: Data Out
   RUNG wire#powerrail
      Contact( #V.RestSolenoid )
      Coil( #DataOut.RestSolenoid )
   END_RUNG
   RUNG wire#powerrail
      Contact( #V.WorkSolenoid )
      Coil( #DataOut.WorkSolenoid )
   END_RUNG
   // the same network as SCL:
   #DataOut.RestSolenoid := #V.RestSolenoid;
   #DataOut.WorkSolenoid := #V.WorkSolenoid;
END_REGION

REGION Network 17: <<< MACHINE STATUS >>>
END_REGION

REGION Network 18: Standstill
   RUNG wire#powerrail
      Contact( #V.ValveSts.StandStill )
      wire#w1
      Coil( #Sts.Standstill )
   END_RUNG
   RUNG wire#powerrail
      Contact( #DSI.DevicesInSafeState )
   END_RUNG wire#w1
   // the same network as SCL:
   #Sts.Standstill := #V.ValveSts.StandStill OR #DSI.DevicesInSafeState;
END_REGION

REGION Network 19: No pending commands
   RUNG wire#powerrail
      I_Contact( "Sys".FirstPLCCycle )
      I_Contact( #COut.Rest_CheckNext )
      I_Contact( #COut.Work_CheckNext )
      I_Contact( #V.ValveCtrl.MoveRest )
      I_Contact( #V.ValveCtrl.MoveWork )
      { S7_Templates := "time_type := Time" } #TON_NoPendingCmd.TON(pt := T#500ms, et =>)
   END_RUNG
   // the same network as SCL:
   #TON_NoPendingCmd(IN := NOT "Sys".FirstPLCCycle AND NOT #COut.Rest_CheckNext AND NOT #COut.Work_CheckNext AND NOT #V.ValveCtrl.MoveRest AND NOT #V.ValveCtrl.MoveWork,   // TON
                     PT := T#500ms);
END_REGION

REGION Network 20: Warnings presence
   RUNG wire#powerrail
      I_Contact( #Warning.NotAutReady )
      I_Contact( #Warning.PressureRunning_Timeout )
      I_Contact( #Warning.Rest_MissingExtEnable )
      I_Contact( #Warning.Work_MissingExtEnable )
      Not()
      Coil( #Sts.WarningsPresence )
   END_RUNG
   // the same network as SCL:
   #Sts.WarningsPresence := NOT (NOT #Warning.NotAutReady AND NOT #Warning.PressureRunning_Timeout AND NOT #Warning.Rest_MissingExtEnable AND NOT #Warning.Work_MissingExtEnable);
END_REGION

REGION Network 21: Alarms presence
   RUNG wire#powerrail
      I_Contact( #V.ValveSts.AlarmPresence )
      I_Contact( #Cin.ExternalAlarms )
      Not()
      Coil( #Sts.AlarmsPresence )
   END_RUNG
   // the same network as SCL:
   #Sts.AlarmsPresence := NOT (NOT #V.ValveSts.AlarmPresence AND NOT #Cin.ExternalAlarms);
END_REGION

REGION Network 22: Stop aborting
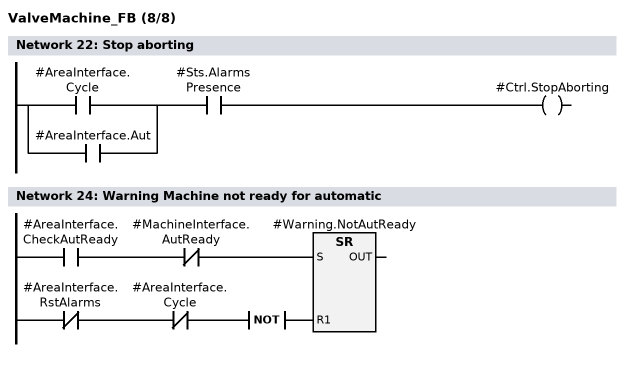
   RUNG wire#powerrail
      Contact( #AreaInterface.Cycle )
      wire#w1
      Contact( #Sts.AlarmsPresence )
      Coil( #Ctrl.StopAborting )
   END_RUNG
   RUNG wire#powerrail
      Contact( #AreaInterface.Aut )
   END_RUNG wire#w1
   // the same network as SCL:
   #Ctrl.StopAborting := (#AreaInterface.Cycle OR #AreaInterface.Aut) AND #Sts.AlarmsPresence;
END_REGION

REGION Network 23 (SCL): Collect machine to zone interface
   #MachineInterface.AutReady := #AreaInterface.Aut AND NOT #Sts.AlarmsPresence;
   #MachineInterface.Aborting := #Ctrl.StopAborting;
   #MachineInterface.MotionsStandStill := #TON_NoPendingCmd.Q AND #Sts.Standstill;
   #MachineInterface.AckStopInPhase := #Ctrl.StopInPhase AND #MachineInterface.MotionsStandStill;
   #MachineInterface.AckStopProgrammed := #Ctrl.StopProgrammed AND #MachineInterface.MotionsStandStill;
   #MachineInterface.AlarmsPresence := #Sts.AlarmsPresence;
   #MachineInterface.WarningPresence := #Sts.WarningsPresence;
END_REGION

REGION Network 24: Warning Machine not ready for automatic
   RUNG wire#powerrail
      Contact( #AreaInterface.CheckAutReady )
      I_Contact( #MachineInterface.AutReady )
      S_SR(operand := #Warning.NotAutReady, r1 := wire#w1)
   END_RUNG
   RUNG wire#powerrail
      I_Contact( #AreaInterface.RstAlarms )
      I_Contact( #AreaInterface.Cycle )
      Not()
   END_RUNG wire#w1
   // the same network as SCL:
   IF #AreaInterface.CheckAutReady AND NOT #MachineInterface.AutReady THEN
       #Warning.NotAutReady := TRUE;   // SR flip-flop
   END_IF;
   IF NOT (NOT #AreaInterface.RstAlarms AND NOT #AreaInterface.Cycle) THEN
       #Warning.NotAutReady := FALSE;
   END_IF;
END_REGION

REGION Network 25 (SCL): ENO
   ENO := NOT #Sts.AlarmsPresence;
END_REGION
END_FUNCTION_BLOCK
